// TIA Portal project "PLC_ThuyKhi_Project" (V16)

(* hardware
DEVICE "S7300/ET200M station_1"  S7-300 station
   slot 0: "Rail_0"  Rail  6ES7 390-1***0-0AA0
   slot 2: "PLC_1"  CPU 314C-2 PN/DP  6ES7 314-6EH04-0AB0  V3.3
      slot 2: "PROFINET interface_1"  PN-IO
         slot 1: "Port_1"  Port
         slot 2: "Port_2"  Port
      slot 5: "DI 24/DO 16_1"  DI24/DO16
      slot 6: "AI 5/AO 2_1"  AI5/AO2
      slot 7: "Count_1"  Counter
      slot 8: "Positioning_1"  Positioning
*)

// ===== PLC "PLC_1"  CPU 314C-2 PN/DP =====

VAR_GLOBAL   // PLC tag table "Default tag table"
   "AUTO/MAN" AT %I0.0 : Bool;
   "TEMP" AT %M1.0 : Bool;
   "A1" AT %Q0.0 : Bool;
   "A2" AT %Q0.1 : Bool;
   "RA" AT %I0.1 : Bool;
   "VO" AT %I0.2 : Bool;
   "S1" AT %I1.0 : Bool;
   "S2" AT %I1.1 : Bool;
   "S3" AT %I1.2 : Bool;
   "L" AT %I1.3 : Bool;
   "M" AT %I1.4 : Bool;
   "H" AT %I1.5 : Bool;
   "EMER" AT %I0.3 : Bool;
   "RESET" AT %I0.4 : Bool;
   "ERROR1" AT %Q0.2 : Bool;
   "Tag_1" AT %M50.0 : Bool;
   "Tag_2" AT %M50.1 : Bool;
   "Tag_3" AT %M50.2 : Bool;
   "Tag_4" AT %M50.3 : Bool;
   "Tag_5" AT %M50.4 : Bool;
   "Tag_6" AT %M50.5 : Bool;
   "Tag_7" AT %M60.0 : Bool;
   "ERROR3" AT %Q0.4 : Bool;
   "ERROR2" AT %Q0.3 : Bool;
   "Tag_8" AT %M10.0 : Bool;
   "Tag_l" AT %M40.0 : Bool;
   "Tag_10" AT %M40.1 : Bool;
   "Tag_m" AT %M40.2 : Bool;
   "Tag_h" AT %M40.3 : Bool;
   "Tag_9" AT %M20.0 : Bool;
   "Tag_11" AT %M20.1 : Bool;
   "Tag_12" AT %M20.2 : Bool;
   "Tag_13" AT %M30.0 : Bool;
   "Tag_14" AT %M30.1 : Bool;
   "SS1" AT %I0.5 : Bool;
   "TEMP_SS2" AT %M30.6 : Bool;
   "TEMP_SS3" AT %M30.7 : Bool;
   "TEMP_AUTO" AT %Q31.0 : Bool;
   "TEMP_1" AT %M31.1 : Bool;
   "TEMP_12" AT %M31.2 : Bool;
   "Tag_15" AT %Q0.6 : Bool;
   "Tag_16" AT %Q0.7 : Bool;
   "Clock" AT %M0.5 : Bool;
   "Tag_17" AT %M11.0 : Bool;
   "Tag_18" AT %M11.1 : Bool;
   "Tag_19" AT %M11.2 : Bool;
   "Count_H" AT %MW24 : Int;
   "Count_M" AT %MW26 : Int;
   "Count_L" AT %MW28 : Int;
   "fasle_H" AT %M90.0 : Bool;
   "fasle_M" AT %M90.1 : Bool;
   "fasle_L" AT %M90.2 : Bool;
   "Tag_20" AT %M90.3 : Bool;
END_VAR

VAR_GLOBAL   // PLC tag table "Tag table_1"
   "HIGH" AT %M5.0 : Bool;
   "MEDIUM" AT %M5.1 : Bool;
   "LOW" AT %M5.2 : Bool;
   "TEMP_H" AT %M5.3 : Bool;
   "TEMP_M" AT %M5.4 : Bool;
   "TEMP_L" AT %M5.5 : Bool;
   "P_H" AT %M5.6 : Bool;
   "P_M" AT %M5.7 : Bool;
   "P_L" AT %M6.0 : Bool;
   "DM_L" AT %M6.1 : Bool;
   "DM_M" AT %M6.2 : Bool;
   "DM_H" AT %M6.3 : Bool;
   "TEMP1" AT %M8.0 : Bool;
   "TEMP2" AT %M8.1 : Bool;
   "TEMP3" AT %M8.2 : Bool;
   "TEMP4" AT %M8.3 : Bool;
   "TEMP5" AT %M8.4 : Bool;
   "TEMP6" AT %M8.5 : Bool;
   "TEMP7" AT %M8.6 : Bool;
   "TEMP8" AT %M8.7 : Bool;
   "T_H" AT %M6.4 : Bool;
   "T_M" AT %M6.5 : Bool;
   "T_L" AT %M6.6 : Bool;
   "TEMP10" AT %M9.0 : Bool;
   "ET_L" AT %MD9 : Time;
   "TEST" AT %MD14 : Time;
   "TEMP11" AT %M13.0 : Bool;
   "TEMP12" AT %M13.1 : Bool;
   "ET_M" AT %MD18 : Time;
   "ET_H" AT %MD22 : Time;
   "TEMP_SS1" AT %M30.2 : Bool;
END_VAR

FUNCTION "FC_RESET" : Void   // FC1, LAD
{ S7_Optimized_Access := 'FALSE' }
VERSION : 0.1
   VAR_TEMP   // added for the SCL form of the ladder/FBD networks
      _w1 : Bool;
   END_VAR
BEGIN

REGION Network 1
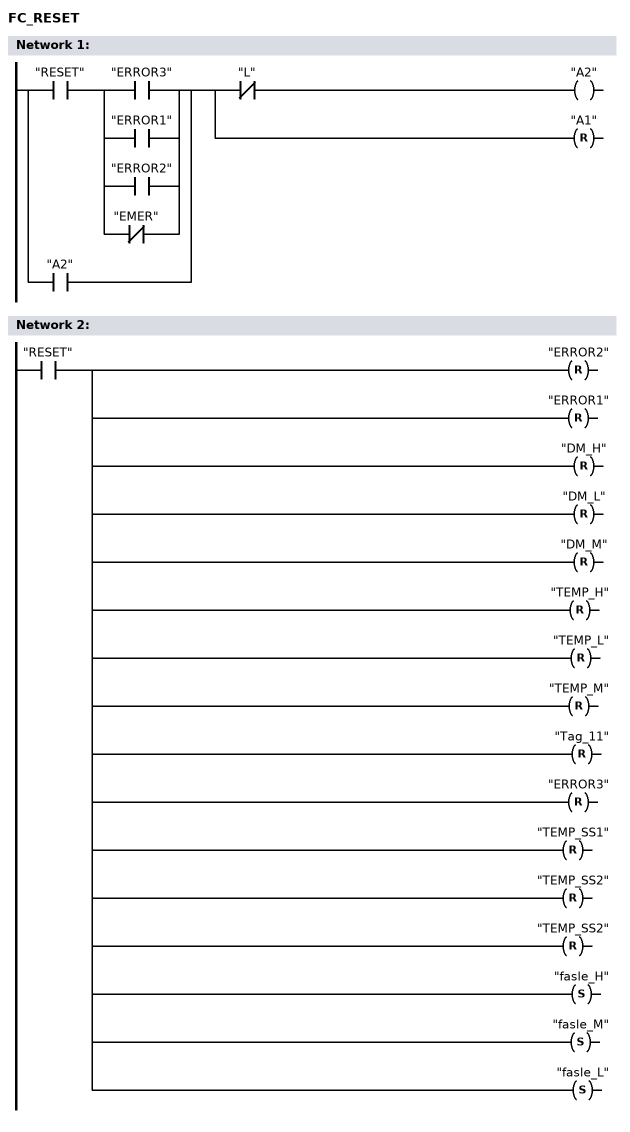
   RUNG wire#powerrail
      Contact( "RESET" )
      wire#w1
      Contact( "ERROR3" )
      wire#w2
      I_Contact( "L" )
      Coil( "A2" )
   END_RUNG
   RUNG wire#w1
      Contact( "ERROR1" )
   END_RUNG wire#w2
   RUNG wire#w1
      Contact( "ERROR2" )
   END_RUNG wire#w2
   RUNG wire#w1
      I_Contact( "EMER" )
   END_RUNG wire#w2
   RUNG wire#powerrail
      Contact( "A2" )
   END_RUNG wire#w2
   RUNG wire#w2
      R_Coil( "A1" )
   END_RUNG
   // the same network as SCL:
   #_w1 := ("RESET" AND ("ERROR3" OR "ERROR1" OR "ERROR2" OR NOT "EMER")) OR "A2";
   "A2" := #_w1 AND NOT "L";
   IF #_w1 THEN "A1" := FALSE; END_IF;
END_REGION

REGION Network 2
   RUNG wire#powerrail
      Contact( "RESET" )
      wire#w1
      R_Coil( "ERROR2" )
   END_RUNG
   RUNG wire#w1
      R_Coil( "ERROR1" )
   END_RUNG
   RUNG wire#w1
      R_Coil( "DM_H" )
   END_RUNG
   RUNG wire#w1
      R_Coil( "DM_L" )
   END_RUNG
   RUNG wire#w1
      R_Coil( "DM_M" )
   END_RUNG
   RUNG wire#w1
      R_Coil( "TEMP_H" )
   END_RUNG
   RUNG wire#w1
      R_Coil( "TEMP_L" )
   END_RUNG
   RUNG wire#w1
      R_Coil( "TEMP_M" )
   END_RUNG
   RUNG wire#w1
      R_Coil( "Tag_11" )
   END_RUNG
   RUNG wire#w1
      R_Coil( "ERROR3" )
   END_RUNG
   RUNG wire#w1
      R_Coil( "TEMP_SS1" )
   END_RUNG
   RUNG wire#w1
      R_Coil( "TEMP_SS2" )
   END_RUNG
   RUNG wire#w1
      R_Coil( "TEMP_SS2" )
   END_RUNG
   RUNG wire#w1
      S_Coil( "fasle_H" )
   END_RUNG
   RUNG wire#w1
      S_Coil( "fasle_M" )
   END_RUNG
   RUNG wire#w1
      S_Coil( "fasle_L" )
   END_RUNG
   // the same network as SCL:
   IF "RESET" THEN
       "ERROR2" := FALSE;
       "ERROR1" := FALSE;
       "DM_H" := FALSE;
       "DM_L" := FALSE;
       "DM_M" := FALSE;
       "TEMP_H" := FALSE;
       "TEMP_L" := FALSE;
       "TEMP_M" := FALSE;
       "Tag_11" := FALSE;
       "ERROR3" := FALSE;
       "TEMP_SS1" := FALSE;
       "TEMP_SS2" := FALSE;
       "TEMP_SS2" := FALSE;
       "fasle_H" := TRUE;
       "fasle_M" := TRUE;
       "fasle_L" := TRUE;
   END_IF;
END_REGION
END_FUNCTION

FUNCTION "Block_1" : Void   // FC2, LAD
{ S7_Optimized_Access := 'FALSE' }
VERSION : 0.1
BEGIN

REGION Network 1
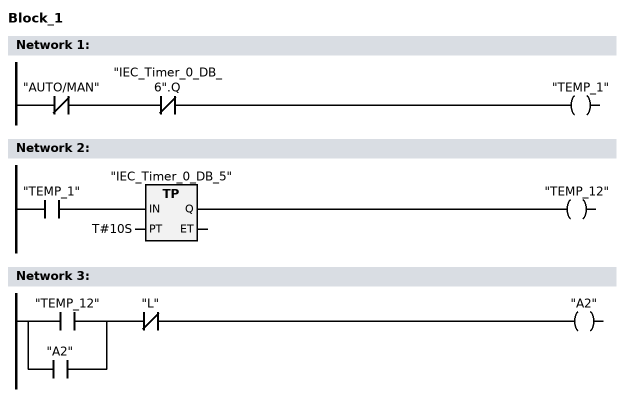
   RUNG wire#powerrail
      I_Contact( "AUTO/MAN" )
      I_Contact( "IEC_Timer_0_DB_6".Q )
      Coil( "TEMP_1" )
   END_RUNG
   // the same network as SCL:
   "TEMP_1" := NOT "AUTO/MAN" AND NOT "IEC_Timer_0_DB_6".Q;
END_REGION

REGION Network 2
   "IEC_Timer_0_DB_5".TP(IN := "TEMP_1", PT := T#10S);
   "TEMP_12" := "IEC_Timer_0_DB_5".Q;
END_REGION

REGION Network 3
   RUNG wire#powerrail
      Contact( "TEMP_12" )
      wire#w1
      I_Contact( "L" )
      Coil( "A2" )
   END_RUNG
   RUNG wire#powerrail
      Contact( "A2" )
   END_RUNG wire#w1
   // the same network as SCL:
   "A2" := ("TEMP_12" OR "A2") AND NOT "L";
END_REGION
END_FUNCTION

FUNCTION "FC_E1_1" : Void   // FC3, LAD
{ S7_Optimized_Access := 'FALSE' }
VERSION : 0.1
   VAR_TEMP   // added for the SCL form of the ladder/FBD networks
      _w1 : Bool;
   END_VAR
BEGIN

REGION Network 1
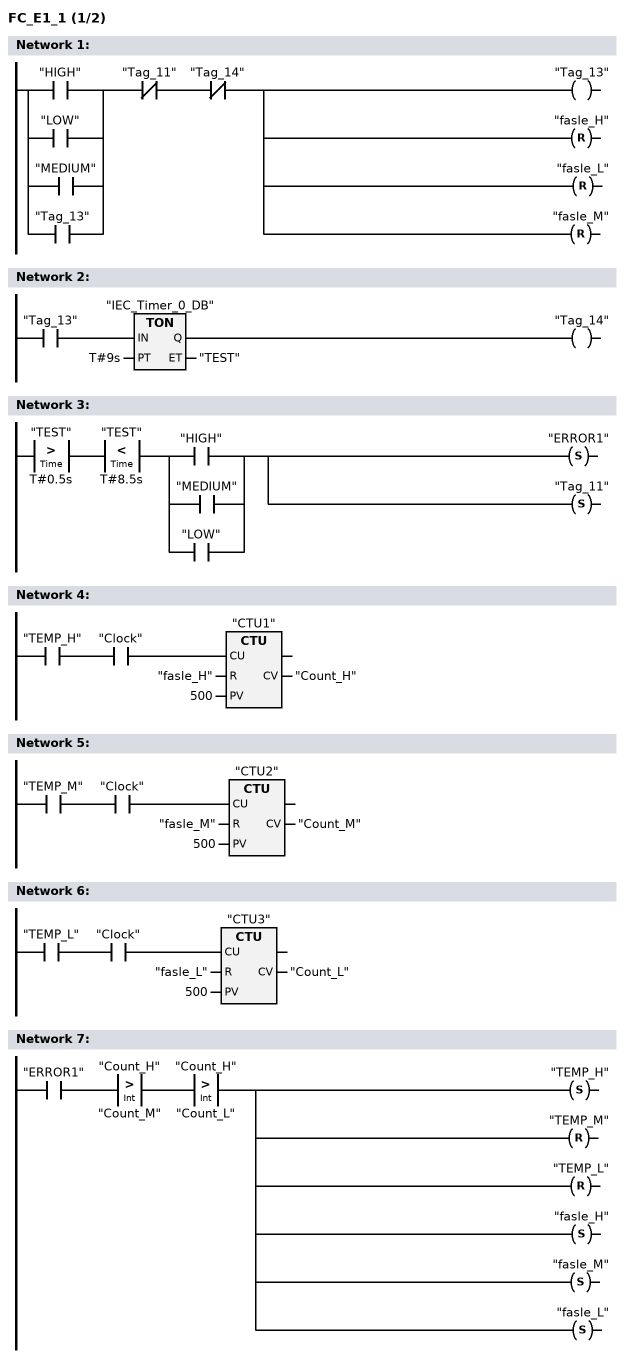
   RUNG wire#powerrail
      Contact( "HIGH" )
      wire#w1
      I_Contact( "Tag_11" )
      I_Contact( "Tag_14" )
      wire#w2
      Coil( "Tag_13" )
   END_RUNG
   RUNG wire#powerrail
      Contact( "LOW" )
   END_RUNG wire#w1
   RUNG wire#powerrail
      Contact( "MEDIUM" )
   END_RUNG wire#w1
   RUNG wire#powerrail
      Contact( "Tag_13" )
   END_RUNG wire#w1
   RUNG wire#w2
      R_Coil( "fasle_H" )
   END_RUNG
   RUNG wire#w2
      R_Coil( "fasle_L" )
   END_RUNG
   RUNG wire#w2
      R_Coil( "fasle_M" )
   END_RUNG
   // the same network as SCL:
   "Tag_13" := ("HIGH" OR "LOW" OR "MEDIUM" OR "Tag_13") AND NOT "Tag_11" AND NOT "Tag_14";
   IF "Tag_13" THEN
       "fasle_H" := FALSE;
       "fasle_L" := FALSE;
       "fasle_M" := FALSE;
   END_IF;
END_REGION

REGION Network 2
   "IEC_Timer_0_DB".TON(IN := "Tag_13", PT := T#9s, ET => "TEST");
   "Tag_14" := "IEC_Timer_0_DB".Q;
END_REGION

REGION Network 3
   RUNG wire#powerrail
      { S7_Templates := "SrcType := Time" } GT_Contact(in1 := "TEST", in2 := T#0.5s)
      { S7_Templates := "SrcType := Time" } LT_Contact(in1 := "TEST", in2 := T#8.5s)
      wire#w1
      Contact( "HIGH" )
      wire#w2
      S_Coil( "ERROR1" )
   END_RUNG
   RUNG wire#w1
      Contact( "MEDIUM" )
   END_RUNG wire#w2
   RUNG wire#w1
      Contact( "LOW" )
   END_RUNG wire#w2
   RUNG wire#w2
      S_Coil( "Tag_11" )
   END_RUNG
   // the same network as SCL:
   IF ("TEST" > T#0.5s) AND ("TEST" < T#8.5s) AND ("HIGH" OR "MEDIUM" OR "LOW") THEN
       "ERROR1" := TRUE;
       "Tag_11" := TRUE;
   END_IF;
END_REGION

REGION Network 4
   "CTU1".CTU(CU := "TEMP_H" AND "Clock", R := "fasle_H", PV := 500, CV => "Count_H");
END_REGION

REGION Network 5
   "CTU2".CTU(CU := "TEMP_M" AND "Clock", R := "fasle_M", PV := 500, CV => "Count_M");
END_REGION

REGION Network 6
   "CTU3".CTU(CU := "TEMP_L" AND "Clock", R := "fasle_L", PV := 500, CV => "Count_L");
END_REGION

REGION Network 7
   RUNG wire#powerrail
      Contact( "ERROR1" )
      { S7_Templates := "SrcType := Int" } GT_Contact(in1 := "Count_H", in2 := "Count_M")
      { S7_Templates := "SrcType := Int" } GT_Contact(in1 := "Count_H", in2 := "Count_L")
      wire#w1
      S_Coil( "TEMP_H" )
   END_RUNG
   RUNG wire#w1
      R_Coil( "TEMP_M" )
   END_RUNG
   RUNG wire#w1
      R_Coil( "TEMP_L" )
   END_RUNG
   RUNG wire#w1
      S_Coil( "fasle_H" )
   END_RUNG
   RUNG wire#w1
      S_Coil( "fasle_M" )
   END_RUNG
   RUNG wire#w1
      S_Coil( "fasle_L" )
   END_RUNG
   // the same network as SCL:
   IF "ERROR1" AND ("Count_H" > "Count_M") AND ("Count_H" > "Count_L") THEN
       "TEMP_H" := TRUE;
       "TEMP_M" := FALSE;
       "TEMP_L" := FALSE;
       "fasle_H" := TRUE;
       "fasle_M" := TRUE;
       "fasle_L" := TRUE;
   END_IF;
END_REGION

REGION Network 8
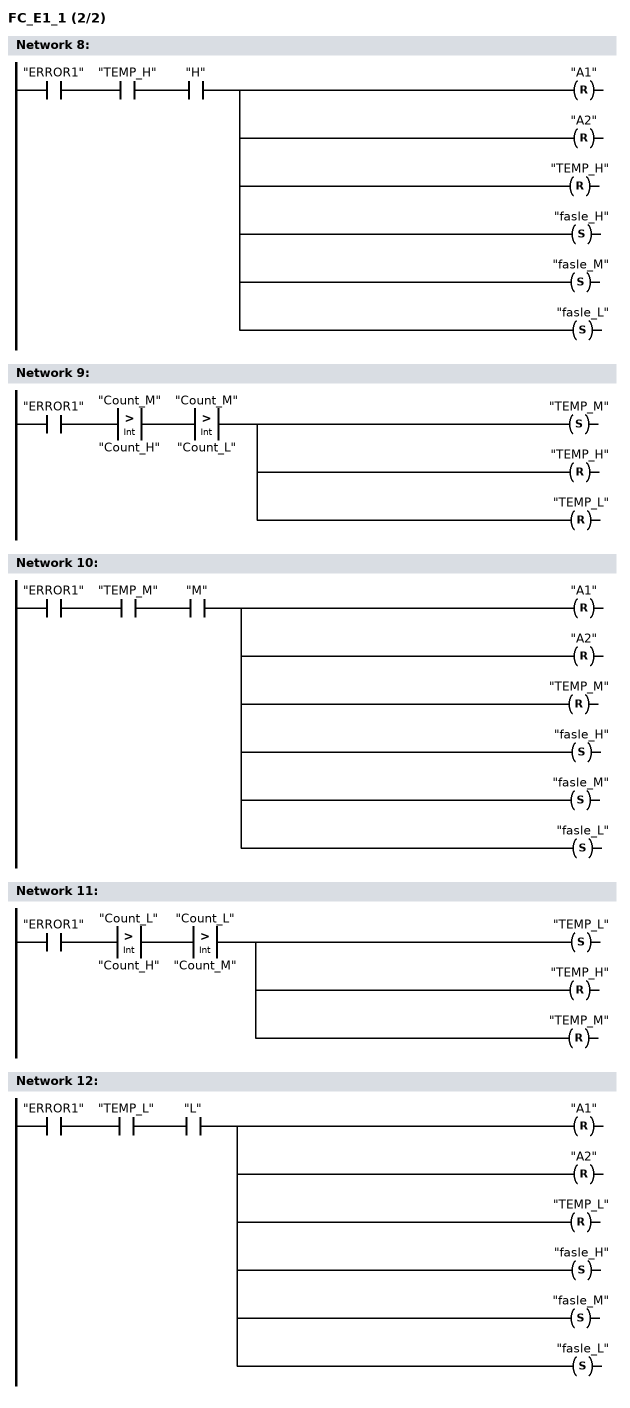
   RUNG wire#powerrail
      Contact( "ERROR1" )
      Contact( "TEMP_H" )
      Contact( "H" )
      wire#w1
      R_Coil( "A1" )
   END_RUNG
   RUNG wire#w1
      R_Coil( "A2" )
   END_RUNG
   RUNG wire#w1
      R_Coil( "TEMP_H" )
   END_RUNG
   RUNG wire#w1
      S_Coil( "fasle_H" )
   END_RUNG
   RUNG wire#w1
      S_Coil( "fasle_M" )
   END_RUNG
   RUNG wire#w1
      S_Coil( "fasle_L" )
   END_RUNG
   // the same network as SCL:
   IF "ERROR1" AND "TEMP_H" AND "H" THEN
       "A1" := FALSE;
       "A2" := FALSE;
   END_IF;
   #_w1 := "ERROR1" AND "TEMP_H" AND "H";
   IF #_w1 THEN
       "TEMP_H" := FALSE;
       "fasle_H" := TRUE;
       "fasle_M" := TRUE;
       "fasle_L" := TRUE;
   END_IF;
END_REGION

REGION Network 9
   RUNG wire#powerrail
      Contact( "ERROR1" )
      { S7_Templates := "SrcType := Int" } GT_Contact(in1 := "Count_M", in2 := "Count_H")
      { S7_Templates := "SrcType := Int" } GT_Contact(in1 := "Count_M", in2 := "Count_L")
      wire#w1
      S_Coil( "TEMP_M" )
   END_RUNG
   RUNG wire#w1
      R_Coil( "TEMP_H" )
   END_RUNG
   RUNG wire#w1
      R_Coil( "TEMP_L" )
   END_RUNG
   // the same network as SCL:
   IF "ERROR1" AND ("Count_M" > "Count_H") AND ("Count_M" > "Count_L") THEN
       "TEMP_M" := TRUE;
       "TEMP_H" := FALSE;
       "TEMP_L" := FALSE;
   END_IF;
END_REGION

REGION Network 10
   RUNG wire#powerrail
      Contact( "ERROR1" )
      Contact( "TEMP_M" )
      Contact( "M" )
      wire#w1
      R_Coil( "A1" )
   END_RUNG
   RUNG wire#w1
      R_Coil( "A2" )
   END_RUNG
   RUNG wire#w1
      R_Coil( "TEMP_M" )
   END_RUNG
   RUNG wire#w1
      S_Coil( "fasle_H" )
   END_RUNG
   RUNG wire#w1
      S_Coil( "fasle_M" )
   END_RUNG
   RUNG wire#w1
      S_Coil( "fasle_L" )
   END_RUNG
   // the same network as SCL:
   IF "ERROR1" AND "TEMP_M" AND "M" THEN
       "A1" := FALSE;
       "A2" := FALSE;
   END_IF;
   #_w1 := "ERROR1" AND "TEMP_M" AND "M";
   IF #_w1 THEN
       "TEMP_M" := FALSE;
       "fasle_H" := TRUE;
       "fasle_M" := TRUE;
       "fasle_L" := TRUE;
   END_IF;
END_REGION

REGION Network 11
   RUNG wire#powerrail
      Contact( "ERROR1" )
      { S7_Templates := "SrcType := Int" } GT_Contact(in1 := "Count_L", in2 := "Count_H")
      { S7_Templates := "SrcType := Int" } GT_Contact(in1 := "Count_L", in2 := "Count_M")
      wire#w1
      S_Coil( "TEMP_L" )
   END_RUNG
   RUNG wire#w1
      R_Coil( "TEMP_H" )
   END_RUNG
   RUNG wire#w1
      R_Coil( "TEMP_M" )
   END_RUNG
   // the same network as SCL:
   IF "ERROR1" AND ("Count_L" > "Count_H") AND ("Count_L" > "Count_M") THEN
       "TEMP_L" := TRUE;
       "TEMP_H" := FALSE;
       "TEMP_M" := FALSE;
   END_IF;
END_REGION

REGION Network 12
   RUNG wire#powerrail
      Contact( "ERROR1" )
      Contact( "TEMP_L" )
      Contact( "L" )
      wire#w1
      R_Coil( "A1" )
   END_RUNG
   RUNG wire#w1
      R_Coil( "A2" )
   END_RUNG
   RUNG wire#w1
      R_Coil( "TEMP_L" )
   END_RUNG
   RUNG wire#w1
      S_Coil( "fasle_H" )
   END_RUNG
   RUNG wire#w1
      S_Coil( "fasle_M" )
   END_RUNG
   RUNG wire#w1
      S_Coil( "fasle_L" )
   END_RUNG
   // the same network as SCL:
   IF "ERROR1" AND "TEMP_L" AND "L" THEN
       "A1" := FALSE;
       "A2" := FALSE;
   END_IF;
   #_w1 := "ERROR1" AND "TEMP_L" AND "L";
   IF #_w1 THEN
       "TEMP_L" := FALSE;
       "fasle_H" := TRUE;
       "fasle_M" := TRUE;
       "fasle_L" := TRUE;
   END_IF;
END_REGION
END_FUNCTION

FUNCTION "FC_2" : Void   // FC8, LAD
{ S7_Optimized_Access := 'FALSE' }
VERSION : 0.1
BEGIN

REGION Network 1
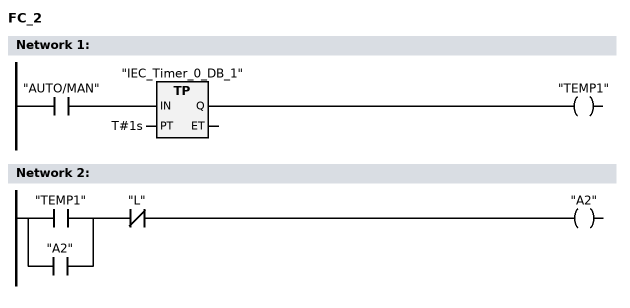
   "IEC_Timer_0_DB_1".TP(IN := "AUTO/MAN", PT := T#1s);
   "TEMP1" := "IEC_Timer_0_DB_1".Q;
END_REGION

REGION Network 2
   RUNG wire#powerrail
      Contact( "TEMP1" )
      wire#w1
      I_Contact( "L" )
      Coil( "A2" )
   END_RUNG
   RUNG wire#powerrail
      Contact( "A2" )
   END_RUNG wire#w1
   // the same network as SCL:
   "A2" := ("TEMP1" OR "A2") AND NOT "L";
END_REGION
END_FUNCTION

FUNCTION "FC_AUTO_1" : Void   // FC9, LAD
{ S7_Optimized_Access := 'FALSE' }
VERSION : 0.1
   VAR_TEMP   // added for the SCL form of the ladder/FBD networks
      _w1 : Bool;
   END_VAR
BEGIN

REGION Network 1
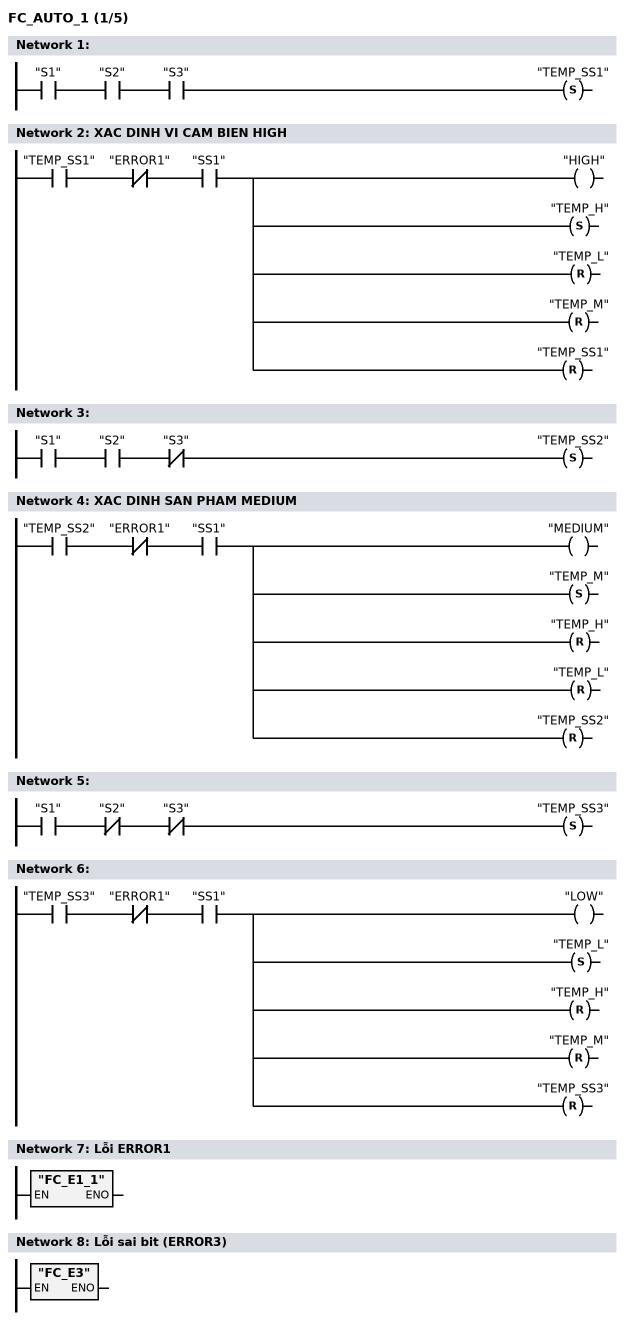
   RUNG wire#powerrail
      Contact( "S1" )
      Contact( "S2" )
      Contact( "S3" )
      S_Coil( "TEMP_SS1" )
   END_RUNG
   // the same network as SCL:
   IF "S1" AND "S2" AND "S3" THEN "TEMP_SS1" := TRUE; END_IF;
END_REGION

REGION Network 2: XAC DINH VI CAM BIEN HIGH
   RUNG wire#powerrail
      Contact( "TEMP_SS1" )
      I_Contact( "ERROR1" )
      Contact( "SS1" )
      wire#w1
      Coil( "HIGH" )
   END_RUNG
   RUNG wire#w1
      S_Coil( "TEMP_H" )
   END_RUNG
   RUNG wire#w1
      R_Coil( "TEMP_L" )
   END_RUNG
   RUNG wire#w1
      R_Coil( "TEMP_M" )
   END_RUNG
   RUNG wire#w1
      R_Coil( "TEMP_SS1" )
   END_RUNG
   // the same network as SCL:
   "HIGH" := "TEMP_SS1" AND NOT "ERROR1" AND "SS1";
   IF "HIGH" THEN
       "TEMP_H" := TRUE;
       "TEMP_L" := FALSE;
       "TEMP_M" := FALSE;
       "TEMP_SS1" := FALSE;
   END_IF;
END_REGION

REGION Network 3
   RUNG wire#powerrail
      Contact( "S1" )
      Contact( "S2" )
      I_Contact( "S3" )
      S_Coil( "TEMP_SS2" )
   END_RUNG
   // the same network as SCL:
   IF "S1" AND "S2" AND NOT "S3" THEN "TEMP_SS2" := TRUE; END_IF;
END_REGION

REGION Network 4: XAC DINH SAN PHAM MEDIUM
   RUNG wire#powerrail
      Contact( "TEMP_SS2" )
      I_Contact( "ERROR1" )
      Contact( "SS1" )
      wire#w1
      Coil( "MEDIUM" )
   END_RUNG
   RUNG wire#w1
      S_Coil( "TEMP_M" )
   END_RUNG
   RUNG wire#w1
      R_Coil( "TEMP_H" )
   END_RUNG
   RUNG wire#w1
      R_Coil( "TEMP_L" )
   END_RUNG
   RUNG wire#w1
      R_Coil( "TEMP_SS2" )
   END_RUNG
   // the same network as SCL:
   "MEDIUM" := "TEMP_SS2" AND NOT "ERROR1" AND "SS1";
   IF "MEDIUM" THEN
       "TEMP_M" := TRUE;
       "TEMP_H" := FALSE;
       "TEMP_L" := FALSE;
       "TEMP_SS2" := FALSE;
   END_IF;
END_REGION

REGION Network 5
   RUNG wire#powerrail
      Contact( "S1" )
      I_Contact( "S2" )
      I_Contact( "S3" )
      S_Coil( "TEMP_SS3" )
   END_RUNG
   // the same network as SCL:
   IF "S1" AND NOT "S2" AND NOT "S3" THEN "TEMP_SS3" := TRUE; END_IF;
END_REGION

REGION Network 6
   RUNG wire#powerrail
      Contact( "TEMP_SS3" )
      I_Contact( "ERROR1" )
      Contact( "SS1" )
      wire#w1
      Coil( "LOW" )
   END_RUNG
   RUNG wire#w1
      S_Coil( "TEMP_L" )
   END_RUNG
   RUNG wire#w1
      R_Coil( "TEMP_H" )
   END_RUNG
   RUNG wire#w1
      R_Coil( "TEMP_M" )
   END_RUNG
   RUNG wire#w1
      R_Coil( "TEMP_SS3" )
   END_RUNG
   // the same network as SCL:
   "LOW" := "TEMP_SS3" AND NOT "ERROR1" AND "SS1";
   IF "LOW" THEN
       "TEMP_L" := TRUE;
       "TEMP_H" := FALSE;
       "TEMP_M" := FALSE;
       "TEMP_SS3" := FALSE;
   END_IF;
END_REGION

REGION Network 7: Lỗi ERROR1
   RUNG wire#powerrail
      "FC_E1_1"()
   END_RUNG
   // the same network as SCL:
   "FC_E1_1"();
END_REGION

REGION Network 8: Lỗi sai bit (ERROR3)
   RUNG wire#powerrail
      "FC_E3"()
   END_RUNG
   // the same network as SCL:
   "FC_E3"();
END_REGION

REGION Network 9
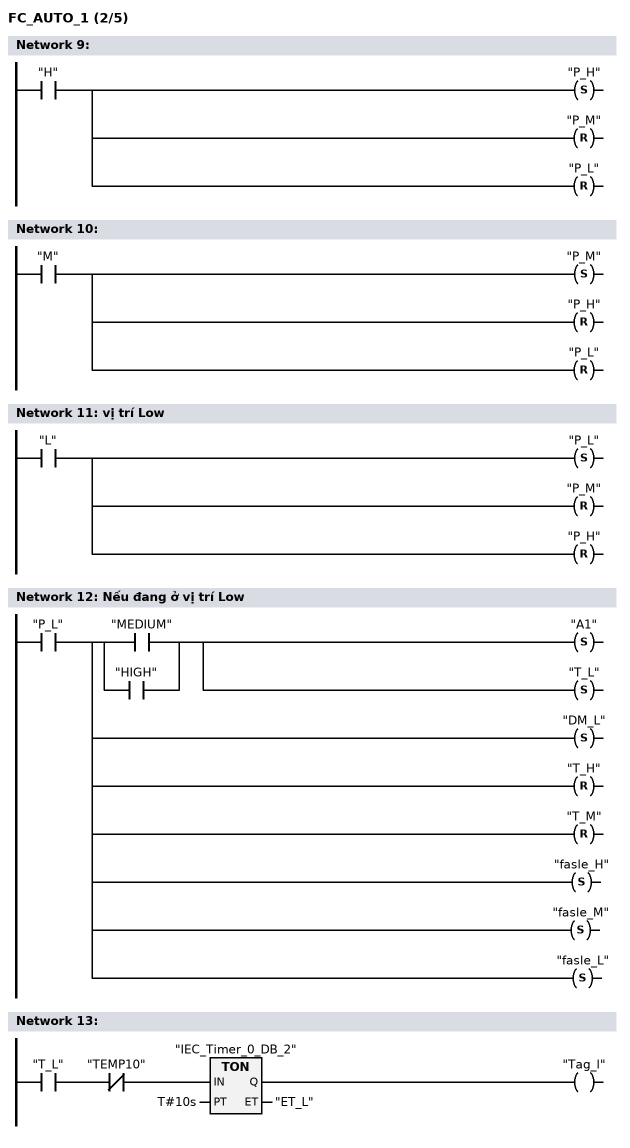
   RUNG wire#powerrail
      Contact( "H" )
      wire#w1
      S_Coil( "P_H" )
   END_RUNG
   RUNG wire#w1
      R_Coil( "P_M" )
   END_RUNG
   RUNG wire#w1
      R_Coil( "P_L" )
   END_RUNG
   // the same network as SCL:
   IF "H" THEN
       "P_H" := TRUE;
       "P_M" := FALSE;
       "P_L" := FALSE;
   END_IF;
END_REGION

REGION Network 10
   RUNG wire#powerrail
      Contact( "M" )
      wire#w1
      S_Coil( "P_M" )
   END_RUNG
   RUNG wire#w1
      R_Coil( "P_H" )
   END_RUNG
   RUNG wire#w1
      R_Coil( "P_L" )
   END_RUNG
   // the same network as SCL:
   IF "M" THEN
       "P_M" := TRUE;
       "P_H" := FALSE;
       "P_L" := FALSE;
   END_IF;
END_REGION

REGION Network 11: vị trí Low
   RUNG wire#powerrail
      Contact( "L" )
      wire#w1
      S_Coil( "P_L" )
   END_RUNG
   RUNG wire#w1
      R_Coil( "P_M" )
   END_RUNG
   RUNG wire#w1
      R_Coil( "P_H" )
   END_RUNG
   // the same network as SCL:
   IF "L" THEN
       "P_L" := TRUE;
       "P_M" := FALSE;
       "P_H" := FALSE;
   END_IF;
END_REGION

REGION Network 12: Nếu đang ở vị trí Low
   RUNG wire#powerrail
      Contact( "P_L" )
      wire#w1
      Contact( "MEDIUM" )
      wire#w2
      S_Coil( "A1" )
   END_RUNG
   RUNG wire#w1
      Contact( "HIGH" )
   END_RUNG wire#w2
   RUNG wire#w2
      S_Coil( "T_L" )
   END_RUNG
   RUNG wire#w1
      S_Coil( "DM_L" )
   END_RUNG
   RUNG wire#w1
      R_Coil( "T_H" )
   END_RUNG
   RUNG wire#w1
      R_Coil( "T_M" )
   END_RUNG
   RUNG wire#w1
      S_Coil( "fasle_H" )
   END_RUNG
   RUNG wire#w1
      S_Coil( "fasle_M" )
   END_RUNG
   RUNG wire#w1
      S_Coil( "fasle_L" )
   END_RUNG
   // the same network as SCL:
   IF "P_L" AND ("MEDIUM" OR "HIGH") THEN
       "A1" := TRUE;
       "T_L" := TRUE;
   END_IF;
   IF "P_L" THEN
       "DM_L" := TRUE;
       "T_H" := FALSE;
       "T_M" := FALSE;
       "fasle_H" := TRUE;
       "fasle_M" := TRUE;
       "fasle_L" := TRUE;
   END_IF;
END_REGION

REGION Network 13
   "IEC_Timer_0_DB_2".TON(IN := "T_L" AND NOT "TEMP10", PT := T#10s, ET => "ET_L");
   "Tag_l" := "IEC_Timer_0_DB_2".Q;
END_REGION

REGION Network 14: Đến quá 5s thì báo lỗi ( cho cả HIGH và MEDIUM), fix cho van tiết lưu 0%
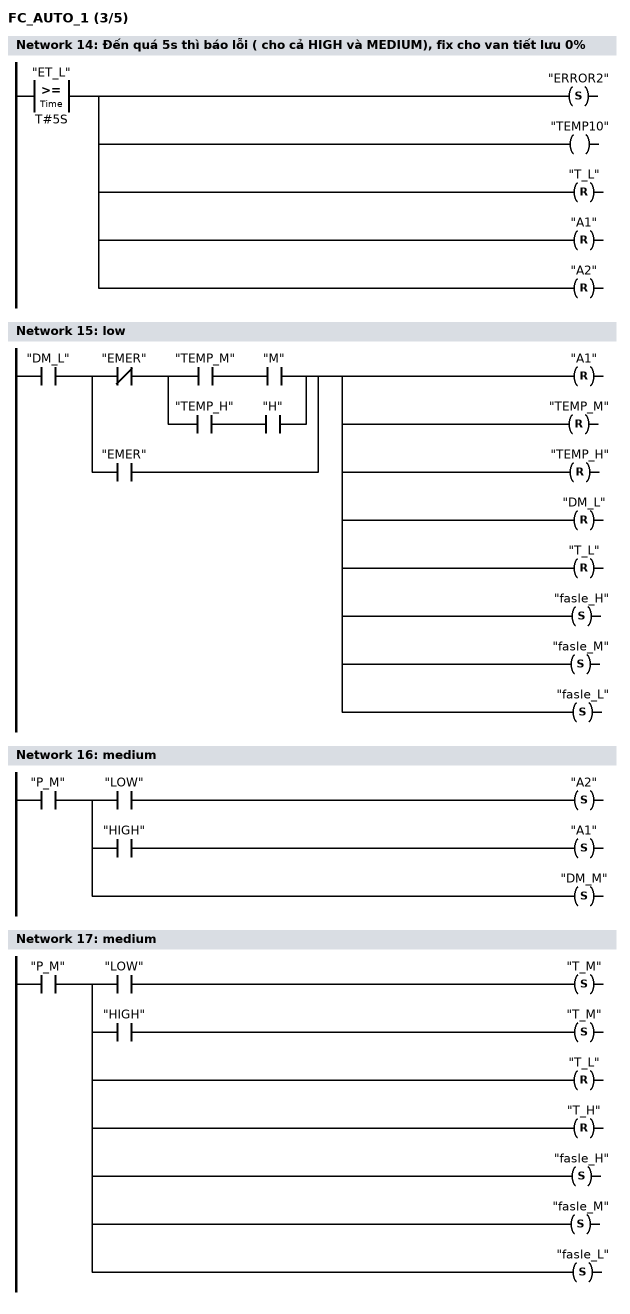
   RUNG wire#powerrail
      { S7_Templates := "SrcType := Time" } GE_Contact(in1 := "ET_L", in2 := T#5S)
      wire#w1
      S_Coil( "ERROR2" )
   END_RUNG
   RUNG wire#w1
      Coil( "TEMP10" )
   END_RUNG
   RUNG wire#w1
      R_Coil( "T_L" )
   END_RUNG
   RUNG wire#w1
      R_Coil( "A1" )
   END_RUNG
   RUNG wire#w1
      R_Coil( "A2" )
   END_RUNG
   // the same network as SCL:
   #_w1 := "ET_L" >= T#5S;
   IF #_w1 THEN "ERROR2" := TRUE; END_IF;
   "TEMP10" := #_w1;
   IF #_w1 THEN
       "T_L" := FALSE;
       "A1" := FALSE;
       "A2" := FALSE;
   END_IF;
END_REGION

REGION Network 15: low
   RUNG wire#powerrail
      Contact( "DM_L" )
      wire#w1
      I_Contact( "EMER" )
      wire#w2
      Contact( "TEMP_M" )
      Contact( "M" )
      wire#w3
      R_Coil( "A1" )
   END_RUNG
   RUNG wire#w2
      Contact( "TEMP_H" )
      Contact( "H" )
   END_RUNG wire#w3
   RUNG wire#w1
      Contact( "EMER" )
   END_RUNG wire#w3
   RUNG wire#w3
      R_Coil( "TEMP_M" )
   END_RUNG
   RUNG wire#w3
      R_Coil( "TEMP_H" )
   END_RUNG
   RUNG wire#w3
      R_Coil( "DM_L" )
   END_RUNG
   RUNG wire#w3
      R_Coil( "T_L" )
   END_RUNG
   RUNG wire#w3
      S_Coil( "fasle_H" )
   END_RUNG
   RUNG wire#w3
      S_Coil( "fasle_M" )
   END_RUNG
   RUNG wire#w3
      S_Coil( "fasle_L" )
   END_RUNG
   // the same network as SCL:
   IF "DM_L" AND ((NOT "EMER" AND (("TEMP_M" AND "M") OR ("TEMP_H" AND "H"))) OR "EMER") THEN
       "A1" := FALSE;
   END_IF;
   #_w1 := "DM_L" AND ((NOT "EMER" AND (("TEMP_M" AND "M") OR ("TEMP_H" AND "H"))) OR "EMER");
   IF #_w1 THEN
       "TEMP_M" := FALSE;
       "TEMP_H" := FALSE;
       "DM_L" := FALSE;
       "T_L" := FALSE;
       "fasle_H" := TRUE;
       "fasle_M" := TRUE;
       "fasle_L" := TRUE;
   END_IF;
END_REGION

REGION Network 16: medium
   RUNG wire#powerrail
      Contact( "P_M" )
      wire#w1
      Contact( "LOW" )
      S_Coil( "A2" )
   END_RUNG
   RUNG wire#w1
      Contact( "HIGH" )
      S_Coil( "A1" )
   END_RUNG
   RUNG wire#w1
      S_Coil( "DM_M" )
   END_RUNG
   // the same network as SCL:
   IF "P_M" AND "LOW" THEN "A2" := TRUE; END_IF;
   IF "P_M" AND "HIGH" THEN "A1" := TRUE; END_IF;
   IF "P_M" THEN "DM_M" := TRUE; END_IF;
END_REGION

REGION Network 17: medium
   RUNG wire#powerrail
      Contact( "P_M" )
      wire#w1
      Contact( "LOW" )
      S_Coil( "T_M" )
   END_RUNG
   RUNG wire#w1
      Contact( "HIGH" )
      S_Coil( "T_M" )
   END_RUNG
   RUNG wire#w1
      R_Coil( "T_L" )
   END_RUNG
   RUNG wire#w1
      R_Coil( "T_H" )
   END_RUNG
   RUNG wire#w1
      S_Coil( "fasle_H" )
   END_RUNG
   RUNG wire#w1
      S_Coil( "fasle_M" )
   END_RUNG
   RUNG wire#w1
      S_Coil( "fasle_L" )
   END_RUNG
   // the same network as SCL:
   IF "P_M" AND "LOW" THEN "T_M" := TRUE; END_IF;
   IF "P_M" AND "HIGH" THEN "T_M" := TRUE; END_IF;
   IF "P_M" THEN
       "T_L" := FALSE;
       "T_H" := FALSE;
       "fasle_H" := TRUE;
       "fasle_M" := TRUE;
       "fasle_L" := TRUE;
   END_IF;
END_REGION

REGION Network 18
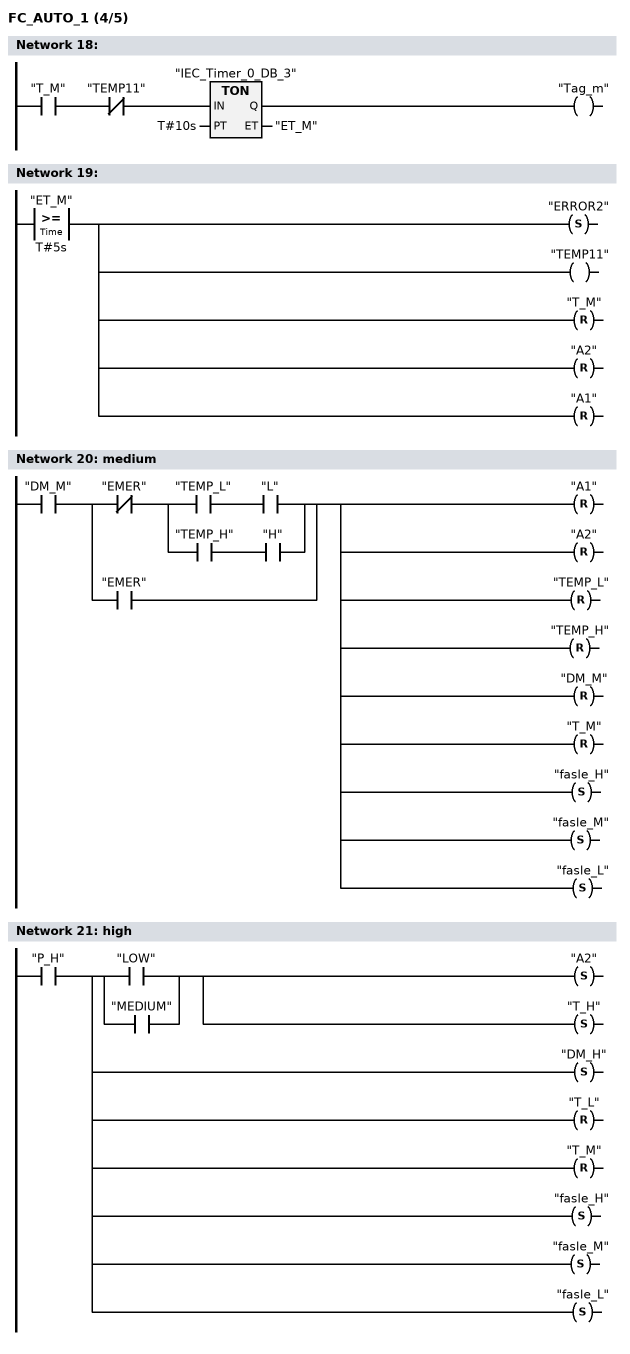
   "IEC_Timer_0_DB_3".TON(IN := "T_M" AND NOT "TEMP11", PT := T#10s, ET => "ET_M");
   "Tag_m" := "IEC_Timer_0_DB_3".Q;
END_REGION

REGION Network 19
   RUNG wire#powerrail
      { S7_Templates := "SrcType := Time" } GE_Contact(in1 := "ET_M", in2 := T#5s)
      wire#w1
      S_Coil( "ERROR2" )
   END_RUNG
   RUNG wire#w1
      Coil( "TEMP11" )
   END_RUNG
   RUNG wire#w1
      R_Coil( "T_M" )
   END_RUNG
   RUNG wire#w1
      R_Coil( "A2" )
   END_RUNG
   RUNG wire#w1
      R_Coil( "A1" )
   END_RUNG
   // the same network as SCL:
   #_w1 := "ET_M" >= T#5s;
   IF #_w1 THEN "ERROR2" := TRUE; END_IF;
   "TEMP11" := #_w1;
   IF #_w1 THEN
       "T_M" := FALSE;
       "A2" := FALSE;
       "A1" := FALSE;
   END_IF;
END_REGION

REGION Network 20: medium
   RUNG wire#powerrail
      Contact( "DM_M" )
      wire#w1
      I_Contact( "EMER" )
      wire#w2
      Contact( "TEMP_L" )
      Contact( "L" )
      wire#w3
      R_Coil( "A1" )
   END_RUNG
   RUNG wire#w2
      Contact( "TEMP_H" )
      Contact( "H" )
   END_RUNG wire#w3
   RUNG wire#w1
      Contact( "EMER" )
   END_RUNG wire#w3
   RUNG wire#w3
      R_Coil( "A2" )
   END_RUNG
   RUNG wire#w3
      R_Coil( "TEMP_L" )
   END_RUNG
   RUNG wire#w3
      R_Coil( "TEMP_H" )
   END_RUNG
   RUNG wire#w3
      R_Coil( "DM_M" )
   END_RUNG
   RUNG wire#w3
      R_Coil( "T_M" )
   END_RUNG
   RUNG wire#w3
      S_Coil( "fasle_H" )
   END_RUNG
   RUNG wire#w3
      S_Coil( "fasle_M" )
   END_RUNG
   RUNG wire#w3
      S_Coil( "fasle_L" )
   END_RUNG
   // the same network as SCL:
   IF "DM_M" AND ((NOT "EMER" AND (("TEMP_L" AND "L") OR ("TEMP_H" AND "H"))) OR "EMER") THEN
       "A1" := FALSE;
       "A2" := FALSE;
   END_IF;
   #_w1 := "DM_M" AND ((NOT "EMER" AND (("TEMP_L" AND "L") OR ("TEMP_H" AND "H"))) OR "EMER");
   IF #_w1 THEN
       "TEMP_L" := FALSE;
       "TEMP_H" := FALSE;
       "DM_M" := FALSE;
       "T_M" := FALSE;
       "fasle_H" := TRUE;
       "fasle_M" := TRUE;
       "fasle_L" := TRUE;
   END_IF;
END_REGION

REGION Network 21: high
   RUNG wire#powerrail
      Contact( "P_H" )
      wire#w1
      Contact( "LOW" )
      wire#w2
      S_Coil( "A2" )
   END_RUNG
   RUNG wire#w1
      Contact( "MEDIUM" )
   END_RUNG wire#w2
   RUNG wire#w2
      S_Coil( "T_H" )
   END_RUNG
   RUNG wire#w1
      S_Coil( "DM_H" )
   END_RUNG
   RUNG wire#w1
      R_Coil( "T_L" )
   END_RUNG
   RUNG wire#w1
      R_Coil( "T_M" )
   END_RUNG
   RUNG wire#w1
      S_Coil( "fasle_H" )
   END_RUNG
   RUNG wire#w1
      S_Coil( "fasle_M" )
   END_RUNG
   RUNG wire#w1
      S_Coil( "fasle_L" )
   END_RUNG
   // the same network as SCL:
   IF "P_H" AND ("LOW" OR "MEDIUM") THEN
       "A2" := TRUE;
       "T_H" := TRUE;
   END_IF;
   IF "P_H" THEN
       "DM_H" := TRUE;
       "T_L" := FALSE;
       "T_M" := FALSE;
       "fasle_H" := TRUE;
       "fasle_M" := TRUE;
       "fasle_L" := TRUE;
   END_IF;
END_REGION

REGION Network 22
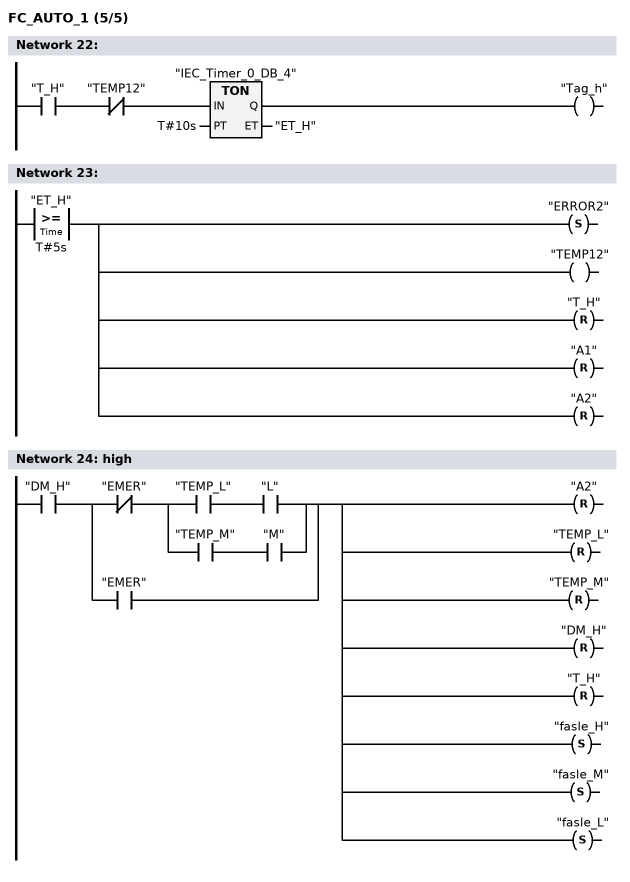
   "IEC_Timer_0_DB_4".TON(IN := "T_H" AND NOT "TEMP12", PT := T#10s, ET => "ET_H");
   "Tag_h" := "IEC_Timer_0_DB_4".Q;
END_REGION

REGION Network 23
   RUNG wire#powerrail
      { S7_Templates := "SrcType := Time" } GE_Contact(in1 := "ET_H", in2 := T#5s)
      wire#w1
      S_Coil( "ERROR2" )
   END_RUNG
   RUNG wire#w1
      Coil( "TEMP12" )
   END_RUNG
   RUNG wire#w1
      R_Coil( "T_H" )
   END_RUNG
   RUNG wire#w1
      R_Coil( "A1" )
   END_RUNG
   RUNG wire#w1
      R_Coil( "A2" )
   END_RUNG
   // the same network as SCL:
   #_w1 := "ET_H" >= T#5s;
   IF #_w1 THEN "ERROR2" := TRUE; END_IF;
   "TEMP12" := #_w1;
   IF #_w1 THEN
       "T_H" := FALSE;
       "A1" := FALSE;
       "A2" := FALSE;
   END_IF;
END_REGION

REGION Network 24: high
   RUNG wire#powerrail
      Contact( "DM_H" )
      wire#w1
      I_Contact( "EMER" )
      wire#w2
      Contact( "TEMP_L" )
      Contact( "L" )
      wire#w3
      R_Coil( "A2" )
   END_RUNG
   RUNG wire#w2
      Contact( "TEMP_M" )
      Contact( "M" )
   END_RUNG wire#w3
   RUNG wire#w1
      Contact( "EMER" )
   END_RUNG wire#w3
   RUNG wire#w3
      R_Coil( "TEMP_L" )
   END_RUNG
   RUNG wire#w3
      R_Coil( "TEMP_M" )
   END_RUNG
   RUNG wire#w3
      R_Coil( "DM_H" )
   END_RUNG
   RUNG wire#w3
      R_Coil( "T_H" )
   END_RUNG
   RUNG wire#w3
      S_Coil( "fasle_H" )
   END_RUNG
   RUNG wire#w3
      S_Coil( "fasle_M" )
   END_RUNG
   RUNG wire#w3
      S_Coil( "fasle_L" )
   END_RUNG
   // the same network as SCL:
   IF "DM_H" AND ((NOT "EMER" AND (("TEMP_L" AND "L") OR ("TEMP_M" AND "M"))) OR "EMER") THEN
       "A2" := FALSE;
   END_IF;
   #_w1 := "DM_H" AND ((NOT "EMER" AND (("TEMP_L" AND "L") OR ("TEMP_M" AND "M"))) OR "EMER");
   IF #_w1 THEN
       "TEMP_L" := FALSE;
       "TEMP_M" := FALSE;
       "DM_H" := FALSE;
       "T_H" := FALSE;
       "fasle_H" := TRUE;
       "fasle_M" := TRUE;
       "fasle_L" := TRUE;
   END_IF;
END_REGION
END_FUNCTION

FUNCTION "FC_MANUAL_1" : Void   // FC10, LAD
{ S7_Optimized_Access := 'FALSE' }
VERSION : 0.1
   VAR_TEMP   // added for the SCL form of the ladder/FBD networks
      _w1 : Bool;
      _w2 : Bool;
      _w3 : Bool;
      _w4 : Bool;
      _w5 : Bool;
      _w6 : Bool;
   END_VAR
BEGIN

REGION Network 1
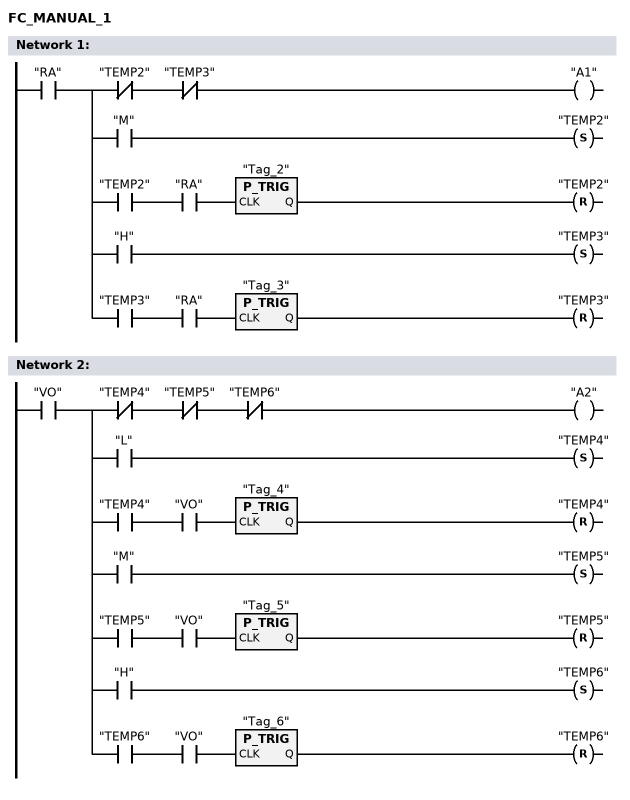
   RUNG wire#powerrail
      Contact( "RA" )
      wire#w1
      I_Contact( "TEMP2" )
      I_Contact( "TEMP3" )
      Coil( "A1" )
   END_RUNG
   RUNG wire#w1
      Contact( "M" )
      S_Coil( "TEMP2" )
   END_RUNG
   RUNG wire#w1
      Contact( "TEMP2" )
      Contact( "RA" )
      P_Trig( "Tag_2" )
      R_Coil( "TEMP2" )
   END_RUNG
   RUNG wire#w1
      Contact( "H" )
      S_Coil( "TEMP3" )
   END_RUNG
   RUNG wire#w1
      Contact( "TEMP3" )
      Contact( "RA" )
      P_Trig( "Tag_3" )
      R_Coil( "TEMP3" )
   END_RUNG
   // the same network as SCL:
   "A1" := "RA" AND NOT "TEMP2" AND NOT "TEMP3";
   IF "RA" AND "M" THEN "TEMP2" := TRUE; END_IF;
   #_w1 := "RA" AND "TEMP2" AND "RA";
   #_w2 := #_w1 AND NOT "Tag_2";   // rising edge
   "Tag_2" := #_w1;
   IF #_w2 THEN "TEMP2" := FALSE; END_IF;
   IF "RA" AND "H" THEN "TEMP3" := TRUE; END_IF;
   #_w3 := "RA" AND "TEMP3" AND "RA";
   #_w4 := #_w3 AND NOT "Tag_3";   // rising edge
   "Tag_3" := #_w3;
   IF #_w4 THEN "TEMP3" := FALSE; END_IF;
END_REGION

REGION Network 2
   RUNG wire#powerrail
      Contact( "VO" )
      wire#w1
      I_Contact( "TEMP4" )
      I_Contact( "TEMP5" )
      I_Contact( "TEMP6" )
      Coil( "A2" )
   END_RUNG
   RUNG wire#w1
      Contact( "L" )
      S_Coil( "TEMP4" )
   END_RUNG
   RUNG wire#w1
      Contact( "TEMP4" )
      Contact( "VO" )
      P_Trig( "Tag_4" )
      R_Coil( "TEMP4" )
   END_RUNG
   RUNG wire#w1
      Contact( "M" )
      S_Coil( "TEMP5" )
   END_RUNG
   RUNG wire#w1
      Contact( "TEMP5" )
      Contact( "VO" )
      P_Trig( "Tag_5" )
      R_Coil( "TEMP5" )
   END_RUNG
   RUNG wire#w1
      Contact( "H" )
      S_Coil( "TEMP6" )
   END_RUNG
   RUNG wire#w1
      Contact( "TEMP6" )
      Contact( "VO" )
      P_Trig( "Tag_6" )
      R_Coil( "TEMP6" )
   END_RUNG
   // the same network as SCL:
   "A2" := "VO" AND NOT "TEMP4" AND NOT "TEMP5" AND NOT "TEMP6";
   IF "VO" AND "L" THEN "TEMP4" := TRUE; END_IF;
   #_w1 := "VO" AND "TEMP4" AND "VO";
   #_w2 := #_w1 AND NOT "Tag_4";   // rising edge
   "Tag_4" := #_w1;
   IF #_w2 THEN "TEMP4" := FALSE; END_IF;
   IF "VO" AND "M" THEN "TEMP5" := TRUE; END_IF;
   #_w3 := "VO" AND "TEMP5" AND "VO";
   #_w4 := #_w3 AND NOT "Tag_5";   // rising edge
   "Tag_5" := #_w3;
   IF #_w4 THEN "TEMP5" := FALSE; END_IF;
   IF "VO" AND "H" THEN "TEMP6" := TRUE; END_IF;
   #_w5 := "VO" AND "TEMP6" AND "VO";
   #_w6 := #_w5 AND NOT "Tag_6";   // rising edge
   "Tag_6" := #_w5;
   IF #_w6 THEN "TEMP6" := FALSE; END_IF;
END_REGION
END_FUNCTION

FUNCTION "FC_E3" : Void   // FC11, LAD
{ S7_Optimized_Access := 'FALSE' }
VERSION : 0.1
BEGIN

REGION Network 1: XAC DINH VI CAM BIEN HIGH
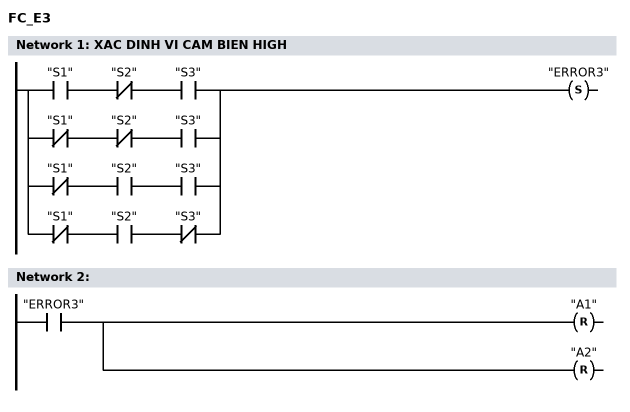
   RUNG wire#powerrail
      Contact( "S1" )
      I_Contact( "S2" )
      Contact( "S3" )
      wire#w1
      S_Coil( "ERROR3" )
   END_RUNG
   RUNG wire#powerrail
      I_Contact( "S1" )
      I_Contact( "S2" )
      Contact( "S3" )
   END_RUNG wire#w1
   RUNG wire#powerrail
      I_Contact( "S1" )
      Contact( "S2" )
      Contact( "S3" )
   END_RUNG wire#w1
   RUNG wire#powerrail
      I_Contact( "S1" )
      Contact( "S2" )
      I_Contact( "S3" )
   END_RUNG wire#w1
   // the same network as SCL:
   IF ("S1" AND NOT "S2" AND "S3") OR (NOT "S1" AND NOT "S2" AND "S3") OR (NOT "S1" AND "S2" AND "S3") OR (NOT "S1" AND "S2" AND NOT "S3") THEN
       "ERROR3" := TRUE;
   END_IF;
END_REGION

REGION Network 2
   RUNG wire#powerrail
      Contact( "ERROR3" )
      wire#w1
      R_Coil( "A1" )
   END_RUNG
   RUNG wire#w1
      R_Coil( "A2" )
   END_RUNG
   // the same network as SCL:
   IF "ERROR3" THEN
       "A1" := FALSE;
       "A2" := FALSE;
   END_IF;
END_REGION
END_FUNCTION

ORGANIZATION_BLOCK "Main"   // OB1, LAD
TITLE = "Main Program Sweep (Cycle)"
{ S7_Optimized_Access := 'FALSE' }
VERSION : 0.1
   VAR_TEMP
      OB1_EV_CLASS : Byte;   // Bits 0-3 = 1 (Coming event), Bits 4-7 = 1 (Event class 1)
      OB1_SCAN_1 : Byte;   // 1 (Cold restart scan 1 of OB 1), 3 (Scan 2-n of OB 1)
      OB1_PRIORITY : Byte;   // Priority of OB Execution
      OB1_OB_NUMBR : Byte;   // 1 (Organization block 1, OB1)
      OB1_RESERVED_1 : Byte;   // Reserved for system
      OB1_RESERVED_2 : Byte;   // Reserved for system
      OB1_PREV_CYCLE : Int;   // Cycle time of previous OB1 scan (milliseconds)
      OB1_MIN_CYCLE : Int;   // Minimum cycle time of OB1 (milliseconds)
      OB1_MAX_CYCLE : Int;   // Maximum cycle time of OB1 (milliseconds)
      OB1_DATE_TIME : Date_And_Time;   // Date and time OB1 started
   END_VAR
   VAR_TEMP   // added for the SCL form of the ladder/FBD networks
      _w1 : Bool;
   END_VAR
BEGIN

REGION Network 1
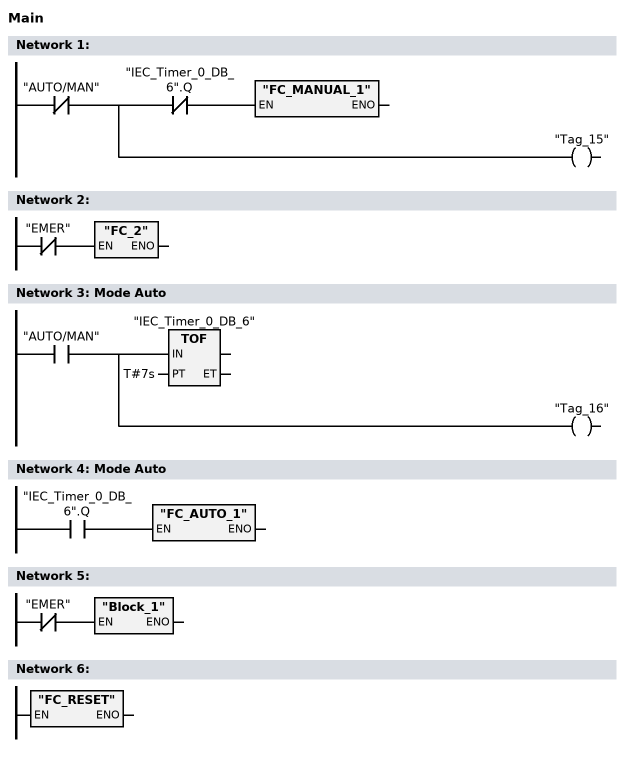
   RUNG wire#powerrail
      I_Contact( "AUTO/MAN" )
      wire#w1
      I_Contact( "IEC_Timer_0_DB_6".Q )
      "FC_MANUAL_1"()
   END_RUNG
   RUNG wire#w1
      Coil( "Tag_15" )
   END_RUNG
   // the same network as SCL:
   #_w1 := NOT "AUTO/MAN";
   IF NOT "AUTO/MAN" AND NOT "IEC_Timer_0_DB_6".Q THEN "FC_MANUAL_1"(); END_IF;
   "Tag_15" := #_w1;
END_REGION

REGION Network 2
   RUNG wire#powerrail
      I_Contact( "EMER" )
      "FC_2"()
   END_RUNG
   // the same network as SCL:
   IF NOT "EMER" THEN "FC_2"(); END_IF;
END_REGION

REGION Network 3: Mode Auto
   "IEC_Timer_0_DB_6".TOF(IN := "AUTO/MAN", PT := T#7s);
   "Tag_16" := "AUTO/MAN";
END_REGION

REGION Network 4: Mode Auto
   RUNG wire#powerrail
      Contact( "IEC_Timer_0_DB_6".Q )
      "FC_AUTO_1"()
   END_RUNG
   // the same network as SCL:
   IF "IEC_Timer_0_DB_6".Q THEN "FC_AUTO_1"(); END_IF;
END_REGION

REGION Network 5
   RUNG wire#powerrail
      I_Contact( "EMER" )
      "Block_1"()
   END_RUNG
   // the same network as SCL:
   IF NOT "EMER" THEN "Block_1"(); END_IF;
END_REGION

REGION Network 6
   RUNG wire#powerrail
      "FC_RESET"()
   END_RUNG
   // the same network as SCL:
   "FC_RESET"();
END_REGION
END_ORGANIZATION_BLOCK